// TIA Portal V20 export
TYPE "UDT_Recipe"
TITLE = Box-product recipe (Module D)
// SCARA Phase 2 Module D recipe (2026-05-23). One flat box-product recipe: product L/W/H + gap, pallet base L/W + layer count, palletizing move dynamics. LPallPatt-shaped (typeProductData / typePalletData / typePnPDynamics, pruned for 1511T -- no block-packing, no mirroring, no interlayers, no multigripper). Consumed by FB_PatternAutoGen, which auto-fits a one-block grid and writes the result into GDB_PalletizingCmd's Module-C config members. PSC binds to GDB_ActiveRecipe.recipe.* member-for-member; the recipe library lives HMI-side on the panel.
   STRUCT
      sName : String[32];   // Recipe name (HMI display / identity).
      bo_Valid : Bool := FALSE;   // PSC handshake: PSC sets FALSE before transferring a parameter set and TRUE only after all members are written. FB_PatternAutoGen consumes the recipe only when this is TRUE -- closes the mid-write race that bites v9's recipe adapter.
      product : Struct
         lr_Length : LReal;   // Box length [mm]. Drives pitchX (= lr_Length + lr_Gap) via FB_PatternAutoGen.
         lr_Width : LReal;   // Box width [mm]. Drives pitchY (= lr_Width + lr_Gap).
         lr_Height : LReal;   // Box height [mm] -- copied straight to GDB_PalletizingCmd.lr_BoxHeight, the layer Z spacing for the Module-C builder.
         lr_Gap : LReal;   // Clearance between boxes [mm]; added to box dims to derive pitch. Set 0 for boxes edge-to-edge.
      END_STRUCT;
      pallet : Struct
         lr_BaseLength : LReal;   // Pallet base length [mm]. FB_PatternAutoGen auto-fits how many boxes fit along X: cols = (BaseLength + Gap) DIV (Length + Gap), floored.
         lr_BaseWidth : LReal;   // Pallet base width [mm]. FB_PatternAutoGen auto-fits how many boxes fit along Y: rows = (BaseWidth + Gap) DIV (Width + Gap), floored.
         i16_LayerCount : Int;   // Stacked layers (tower mode -- all layers use the same auto-gen grid). Total boxes = cols x rows x LayerCount, capped at the GDB_PalletizingPath.aCmd[] ceiling (22 for aCmd[1..200]).
      END_STRUCT;
      dynamics : Struct
         lr_Velocity : LReal;   // Palletizing-move path velocity [mm/s]. Written into GDB_PalletizingCmd.lr_MoveVelocity by FB_PatternAutoGen.
         lr_Acceleration : LReal;   // Palletizing-move acceleration [mm/s^2]. Written into GDB_PalletizingCmd.lr_MoveAccel.
         lr_Deceleration : LReal;   // Palletizing-move deceleration [mm/s^2]. Written into GDB_PalletizingCmd.lr_MoveDecel.
         lr_Jerk : LReal;   // Palletizing-move jerk [mm/s^3]. Written into GDB_PalletizingCmd.lr_MoveJerk.
      END_STRUCT;
   END_STRUCT;
END_TYPE
